VISUALIZATION visuTank  // 2x2
END_VISUALIZATION

(* stored: Version 1.1.0.1, ProductVersion 3.1.4022.17
   Visu visuTank: Id {8c508200-b7fa-4877-b0ce-5135a4901277} *)
